// TIA Portal V20 export
// export: Created 2025-12-01T14:56:14.3963501Z, ExportSetting None, DisplayName Totally Integrated Automation Portal, DisplayVersion V20 Update 3, DisplayName TIA Portal Openness, DisplayVersion V20 Update 3, DisplayName TIA Portal Version Control Interface, DisplayVersion V20 Update 3, DisplayName STEP 7 Professional, DisplayVersion V20 Update 3, DisplayName STEP 7 Safety, DisplayVersion V20 Update 2, DisplayName WinCC Basic/Comfort/Advanced, DisplayVersion V20 Update 3, DisplayName WinCC Professional, DisplayVersion V20 Update 3, DisplayName WinCC Unified, DisplayVersion V20 Update 3
TYPE "UDT_ProtocoloEmiDispositivo"
   STRUCT
      Marcha : Bool;   // El Dispositivo esta en marcha
      Paro : Bool;   // El Dispositivo esta en Paro
      Error : Bool;   // El Dispositivo esta en Error
      Reset_Realizandose : Bool;   // El Dispositivo esta Realizando el Reset
      Automatico : Bool;   // El Dispositivo esta en Automatico
      Mantenimiento : Bool;   // El Dispositivo esta en modo mantenimiento
      Manual : Bool;   // El Dispositivo esta en Manual
      ParoBlando_Realizandose : Bool;   // El Dispositivo esta Realizando el Paro Blando
      ResetNOK : Bool;   // Reset no se ha podido realizar
      ResetOK : Bool;   // Reset se ha realizado
      ParoBlandoNOK : Bool;   // Paro Blando no se ha pordido realizar
      ParoBlandoOK : Bool;   // Paro Blando se ha realizado
      Bit_14 : Bool;
      Bit_15 : Bool;
      Bit_16 : Bool;
      RecepOK : Bool;   // Recepcion OK de la Orden
   END_STRUCT;
END_TYPE
